TYPE EtcSlaveBase_82538BE2 :
STRUCT
END_STRUCT
END_TYPE

(* stored: Version 1.2.0.0, ProductVersion 3.1.4024.12
   DUT EtcSlaveBase_82538BE2: Id {7bd7a308-c04b-0c47-03d6-603e3adab4f5} *)
